SYSTEM hello
  (* Version 1.0, 2022-07-21, alex *)
  APPLICATION helloApp
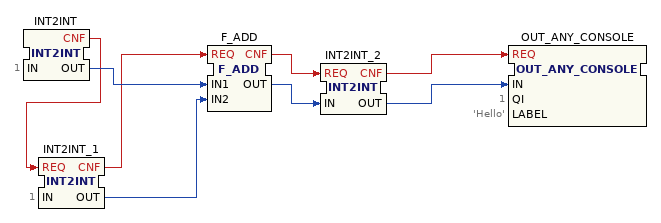
    FBS
      OUT_ANY_CONSOLE : OUT_ANY_CONSOLE(QI := 1, LABEL := 'Hello');
      F_ADD : F_ADD;
      INT2INT : INT2INT(IN := 1);
      INT2INT_1 : INT2INT(IN := 1);
      INT2INT_2 : INT2INT;
    END_FBS
    EVENT_CONNECTIONS
      F_ADD.CNF TO INT2INT_2.REQ;
      INT2INT_2.CNF TO OUT_ANY_CONSOLE.REQ;
      INT2INT.CNF TO INT2INT_1.REQ;
      INT2INT_1.CNF TO F_ADD.REQ;
    END_CONNECTIONS
    DATA_CONNECTIONS
      INT2INT_2.OUT TO OUT_ANY_CONSOLE.IN;
      F_ADD.OUT TO INT2INT_2.IN;
      INT2INT.OUT TO F_ADD.IN1;
      INT2INT_1.OUT TO F_ADD.IN2;
    END_CONNECTIONS
  END_APPLICATION
  DEVICE FORTE_PC : FORTE_PC(MGR_ID := "localhost:61499")
    {SET_ATTRIBUTE(Profile, HOLOBLOC)} (* device profile *)
    RESOURCE EMB_RES : EMB_RES
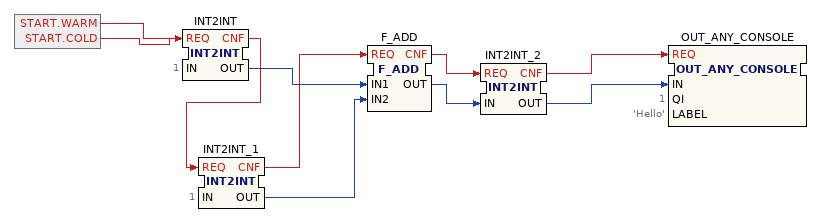
      FBS
        INT2INT : INT2INT(IN := 1);
        INT2INT_1 : INT2INT(IN := 1);
        F_ADD : F_ADD;
        INT2INT_2 : INT2INT;
        OUT_ANY_CONSOLE : OUT_ANY_CONSOLE(QI := 1, LABEL := 'Hello');
      END_FBS
      EVENT_CONNECTIONS
        INT2INT.CNF TO INT2INT_1.REQ;
        INT2INT_1.CNF TO F_ADD.REQ;
        F_ADD.CNF TO INT2INT_2.REQ;
        INT2INT_2.CNF TO OUT_ANY_CONSOLE.REQ;
        START.WARM TO INT2INT.REQ;
        START.COLD TO INT2INT.REQ;
      END_CONNECTIONS
      DATA_CONNECTIONS
        INT2INT.OUT TO F_ADD.IN1;
        INT2INT_1.OUT TO F_ADD.IN2;
        F_ADD.OUT TO INT2INT_2.IN;
        INT2INT_2.OUT TO OUT_ANY_CONSOLE.IN;
      END_CONNECTIONS
    END_RESOURCE
  END_DEVICE
  MAPPINGS
    helloApp.INT2INT ON FORTE_PC.EMB_RES.INT2INT;
    helloApp.INT2INT_1 ON FORTE_PC.EMB_RES.INT2INT_1;
    helloApp.F_ADD ON FORTE_PC.EMB_RES.F_ADD;
    helloApp.INT2INT_2 ON FORTE_PC.EMB_RES.INT2INT_2;
    helloApp.OUT_ANY_CONSOLE ON FORTE_PC.EMB_RES.OUT_ANY_CONSOLE;
  END_MAPPINGS
  SEGMENTS
    Ethernet : Ethernet;
  END_SEGMENTS
  LINKS
    FORTE_PC => Ethernet;
  END_LINKS
END_SYSTEM
